// TwinCAT 3 PLC project Untitled1
// ProgramVersion: 3.1.4024.0
// libraries:
//   SPT Base Types, * (Beckhoff Automation LLC)
//   Tc2_Standard, * (Beckhoff Automation GmbH)
//   Tc2_System, * (Beckhoff Automation GmbH)
//   Tc3_Module, * (Beckhoff Automation GmbH)
//   Tc3_PackML_V2, * (Beckhoff Automation GmbH)
// project tree:
//   / GlobalTextList.TcGTLO, PlcTask.TcTTO, Visualization Manager.TcVMO (not stored)
//   Interfaces/ ITF_Observable.TcIO, ITF_Observer.TcIO
//   POUs/ CD_SPT_EM_Observer.TcCD (not stored), EquipmentModule.TcPOU, MachineModule.TcPOU, MAIN.TcPOU
// real-time tasks:
//   TASK PlcTask: cycle T#10ms, priority 20, ADS port 350

CONFIGURATION Untitled1
    RESOURCE PLC ON TwinCAT3
        TASK PlcTask(INTERVAL := T#10ms, PRIORITY := 20);
        PROGRAM MAIN WITH PlcTask : MAIN;
    END_RESOURCE
END_CONFIGURATION

// ---- Interfaces/ITF_Observable.TcIO
INTERFACE ITF_Observable

METHOD notifyObserver : BOOL
END_METHOD

METHOD registerObserver : BOOL
VAR_INPUT
	Observer : ITF_Observer;
END_VAR
END_METHOD

METHOD removeObserver : BOOL
VAR_INPUT
	Observer : ITF_Observer;
END_VAR
END_METHOD

END_INTERFACE

// ---- Interfaces/ITF_Observer.TcIO
INTERFACE ITF_Observer

METHOD update : BOOL
VAR_INPUT
	Module : REFERENCE TO MachineModule;
END_VAR
END_METHOD

END_INTERFACE

// ---- POUs/MAIN.TcPOU
PROGRAM MAIN
VAR
	Machine : MachineModule := (Name := 'Machine');
END_VAR

Machine.CyclicLogic();

END_PROGRAM

// ---- POUs/MachineModule.TcPOU
FUNCTION_BLOCK MachineModule EXTENDS FB_PackML_BaseModule IMPLEMENTS ITF_Observable
VAR
	//SubModules
	Equip1 : EquipmentModule := (Name := 'EM1');
	Equip2 : EquipmentModule := (Name := 'EM2');
	Equip3 : EquipmentModule := (Name := 'EM3');

	//ITF_Observable
	_Observers : ARRAY[1..Parameters_PackML_Base.MAX_NO_OF_SUBMODULES +1] OF ITF_Observer;

	//Data to be Observered
	_data	 : UDINT;
	dataPrev : UDINT;

	//CyclicLogic
	fbRT	  : R_TRIG;
	register1 : BOOL;
	remove1	  : BOOL;
	register2 : BOOL;
	remove2	  : BOOL;
	register3 : BOOL;
	remove3	  : BOOL;
END_VAR

METHOD PUBLIC CyclicLogic
IF NOT _InitComplete THEN
    _InitComplete := Initialize();
    RETURN;
END_IF

//On data change call all observers
fbRT(CLK:= data <> dataPrev);
IF fbRT.Q THEN
	notifyObserver();
	dataPrev := data;
END_IF


//Attach Observer
IF register1 THEN
	IF 	registerObserver(Equip1) THEN
		register1 := FALSE;
	END_IF
END_IF
IF register2 THEN
	IF 	registerObserver(Equip2) THEN
		register2 := FALSE;
	END_IF
END_IF
IF register3 THEN
	IF 	registerObserver(Equip3) THEN
		register3 := FALSE;
	END_IF
END_IF

//Detach Observer
IF remove1 THEN
	IF removeObserver(Equip1) THEN 
		remove1 := FALSE;
	END_IF
END_IF
IF remove2 THEN
	IF removeObserver(Equip2) THEN 
		remove2 := FALSE;
	END_IF
END_IF
IF remove3 THEN
	IF removeObserver(Equip3) THEN 
		remove3 := FALSE;
	END_IF
END_IF

//Change this value for testing
_data;
END_METHOD

PROPERTY Data : udint
GET
Data := _data;
END_GET
END_PROPERTY

METHOD PROTECTED Initialize : BOOL
Initialize := FALSE;
CASE DescendantSequenceState OF
	0:
		//
		RegisterSubmodule(Equip1);
		RegisterSubmodule(Equip2);
		RegisterSubmodule(Equip3);

		//
		registerObserver(Equip1);
		registerObserver(Equip2);
		registerObserver(Equip3);

		//
		_LogModeChanges			:= FALSE;
		_LogStateChanges		:= FALSE;
		DescendantSequenceState := DescendantSequenceState + 10;

	10:
		(* Call the Super *)
		IF SUPER^.Initialize() THEN
			DescendantSequenceState := DescendantSequenceState + 10;
		END_IF

	20:
		Initialize := TRUE;
END_CASE
END_METHOD

METHOD notifyObserver : BOOL
VAR
	i : UDINT;
END_VAR
//Call all registered Observers and pass them the Observable
FOR i := 1 TO Parameters_PackML_Base.MAX_NO_OF_SUBMODULES DO
	IF _Observers[i] <> 0 THEN
		_Observers[i].update(THIS^);
	END_IF
END_FOR
END_METHOD

METHOD registerObserver : BOOL
VAR_INPUT
	Observer : ITF_Observer;
END_VAR

VAR
	i : UDINT;
END_VAR
registerObserver := FALSE;

//Check if Observer is already registered
FOR i := 1 TO Parameters_PackML_Base.MAX_NO_OF_SUBMODULES DO
	IF _Observers[i] = Observer THEN
		RETURN;
	END_IF
END_FOR

//Add Observer to first available index within the array
FOR i := 1 TO Parameters_PackML_Base.MAX_NO_OF_SUBMODULES DO
	IF _Observers[i] = 0 THEN
		_Observers[i]	 := Observer;
		registerObserver := TRUE;
		EXIT;
	END_IF
END_FOR
END_METHOD

METHOD removeObserver : BOOL
VAR_INPUT
	Observer : ITF_Observer;
END_VAR

VAR
	i : UDINT;
END_VAR
removeObserver := FALSE;

//Check for valid input
IF (Observer = 0) THEN
	RETURN;
END_IF

//Find Observer to be removed and set the array index to 0, will remove duplicates if they exist
FOR i := 1 TO Parameters_PackML_Base.MAX_NO_OF_SUBMODULES DO
	IF (_Observers[i] = Observer) THEN
		_Observers[i]  := 0;
		removeObserver := TRUE;
	END_IF
END_FOR

//Clean up array
FOR i := 1 TO Parameters_PackML_Base.MAX_NO_OF_SUBMODULES DO
	IF _Observers[i] = 0 THEN
		//array size is declared to +1 for these 2 lines of code to be safe
		_Observers[i]	  := _Observers[i + 1];
		_Observers[i + 1] := 0;
	END_IF
END_FOR
END_METHOD

END_FUNCTION_BLOCK

// ---- POUs/EquipmentModule.TcPOU
FUNCTION_BLOCK EquipmentModule EXTENDS FB_PackML_BaseModule IMPLEMENTS ITF_Observer
VAR
	//data from Observable
	data : UDINT;
END_VAR

METHOD PUBLIC CyclicLogic
VAR
	i : UDINT;
END_VAR
IF NOT _InitComplete THEN
	_InitComplete := Initialize();
	RETURN;
END_IF
END_METHOD

METHOD PROTECTED Initialize : BOOL
Initialize := true;
END_METHOD

METHOD update : BOOL
VAR_INPUT
	Module : REFERENCE TO MachineModule;
END_VAR
//Get desired info from Observable
data := Module.Data;
END_METHOD

END_FUNCTION_BLOCK

// ---- GlobalTextList.TcGTLO
TEXTLIST GlobalTextList
  988 = '%i'
  330 = 'EM1: %i'
  363 = 'Equipment Module 1'
  513 = 'Equipment Module 2'
  328 = 'Equipment Module 3'
  542 = 'Register'
END_TEXTLIST
